/// This function block automatically reserves a zone on the window tracking.
/// Remark: Only one zone at the time
FUNCTION_BLOCK FB_TrackingReservation IMPLEMENTS I_TrackingActionListener
(************************************************************************************** 
* 	Application 		: BoxControl Framework 
* 	Revision 			: $Revision: 408723 $ 
* 	Revision date 		: $Date: 2018-06-27 13:49:08 +0200 (Wed, 27 Jun 2018) $ 
* 	Last changed by 	: $Author: b7bolm $ 
* 	URL 				: $URL: http://almscdc.swisslog.com/repo/SWPD/Development/BoxControlFramework/21_Projects/BCF_2.0/trunk/BCF/BCF/JumpStart/20_Product/10_App/12_E_Functions/10_Lib/10_Conv/FB_FunctionList.TcPOU $ 
* ------------------------------------------------------------------------------------ 
* 	© Swisslog AG 
* 	Swisslog is not liable for any usage of this source code that is not agreed 
* 	on between Swisslog and the other party. The mandatory legal liability remains 
* 	unaffected. 
* ------------------------------------------------------------------------------------ 
* 	Revision History: 
* 
* 	VERSION 		DATE 			INITIALS 			DESCRIPTION 
* 	0.1 			25.09.2018 		mbo					First implementation
* 
**************************************************************************************)
VAR_INPUT
	Enable					: BOOL; // Enable reservation
	ActionId				: INT; // Action id for zone
	AbsolutePosition		: DINT; // Position where it should be earliest reserved
	Length					: UINT; // length of tracking zone to be reserved
	MaxDistance				: UDINT; // Max distance in which its allowed to be reserved (0=Full range)
	PositionToLive			: UDINT; // Position after the reserved zones gets deleted if not used
	MinimumDistance			: UINT; // Minimum gap until next reservation [mm]
	iWindowTracking			: I_WindowTracking; // Link to window tracking
END_VAR
VAR_OUTPUT
	ReservedZoneIndex		: UINT; // Currently reserved zone index
END_VAR
VAR
	LastReservedZoneIndex	: UINT; // Last reserved zone index
	LastZoneEndPosition		: UDINT; // Last zone end position
END_VAR

// Check inputs
IF iWindowTracking = 0 OR 
   ActionId = 0 OR
   Length = 0 THEN
	RETURN;
END_IF

// Reserve a new zone if required
IF Enable THEN
	
	IF ReservedZoneIndex = 0 THEN
		LastZoneEndPosition := iWindowTracking.M_GetZoneEndPosition(LastReservedZoneIndex);
		
		IF AbsolutePosition + MinimumDistance < UDINT_TO_DINT(LastZoneEndPosition) OR LastZoneEndPosition = 0 THEN
			ReservedZoneIndex := iWindowTracking.M_AllocateNextFreeZone(
													mActionId 			:= ActionId,
													mAbsolutePosition 	:= DINT_TO_UDINT(AbsolutePosition),
													mLength 			:= Length,
													mMaxDistance 		:= MaxDistance,
													miActionListener 	:= THIS^,
													mPositionToLive 	:= PositionToLive);
		END_IF
	END_IF
END_IF

METHOD M_ActionZoneChangedEvent

VAR_INPUT
	mZoneIndex	: UINT; // Deleted zone index
	mZoneData	: ST_WindowTrackingZone; // Data of deleted zone
END_VAR
// Reset when zone gets occupied
IF mZoneData.TU_Present THEN
	LastReservedZoneIndex := ReservedZoneIndex;
	ReservedZoneIndex := 0;
END_IF
END_METHOD

// Automatically called whenever the stored zone gets deleted on tracking
METHOD M_ActionZoneDeletedEvent
VAR_INPUT
	mZoneIndex	: UINT; //  Deleted zone index
	mZoneData	: ST_WindowTrackingZone; // Data of deleted zone
END_VAR
IF mZoneIndex = ReservedZoneIndex THEN
	ReservedZoneIndex := 0;
	
ELSIF mZoneIndex = LastReservedZoneIndex THEN
	LastReservedZoneIndex := 0;
END_IF
END_METHOD

/// Delete pending reservation
METHOD M_ClearReservation : BOOL // Returns true if successfully deleted
VAR_INPUT
END_VAR
M_ClearReservation := FALSE;

IF iWindowTracking <> 0 THEN
	IF ReservedZoneIndex > 0 THEN
		M_ClearReservation := iWindowTracking.M_DeleteZone(ReservedZoneIndex);
	END_IF
END_IF
END_METHOD

END_FUNCTION_BLOCK

(* stored: Version 1.1.0.1, ProductVersion 3.1.4022.12
   POU FB_TrackingReservation: Id {b5a46420-a8c0-40c8-a792-6ee9f5753ca9}, SpecialFunc None
   Method M_ActionZoneChangedEvent: Id {bd2b7e33-f7f2-405a-bf6b-41c98eabec56}
   Method M_ActionZoneDeletedEvent: Id {9cf3b968-c336-4366-8029-89466eff2a62}
   Method M_ClearReservation: Id {1a3299c6-0a4f-4353-a77a-7e9c6d964951} *)
